// TIA Portal V20 export
TYPE "LBP_typeChanX"
TITLE = Channel interface / Interface de canal
// User data type for blocks LBP_Chan1 [DB21] .. LBP_Chan10 [DB30] / Type de données utilisateur pour les blocs LBP_Chan1 [DB21] .. LBP_Chan10 [DB30]
   STRUCT
      f0_0 : Bool;
      f0_1 : Bool;
      f0_2 : Bool;
      A_DRF : Bool;   // Activate DRF / Activer DRF
      A_SBL : Bool;   // Activate single block / Activer bloc par bloc
      A_M01 : Bool;   // Activate M01 / Activer M01
      A_DRY : Bool;   // Activate dry run feedrate / Activer avance marche d'essai
      f0_7 : Bool;
      A_Ref : Bool;   // Activate referencing / Activer référencement
      A_ProtZone : Bool;   // Enable protection zones / Activer zones de protection
      A_SynOff : Bool;   // Synchronous action off / Action synchrone désactivée
      A_TM_TimOut : Bool;   // Activate time-out (TM) / Activer timeout (TM)
      A_CLC_Stop : Bool;   // CLC stop / Stop CLC
      A_CLC_OR : Bool;   // CLC override / Correction CLC
      A_PLC_ActCompl : Bool;   // PLC action completed / Action AP terminée
      A_ProgTest : Bool;   // Activate program test / Activer test de programme
      A_SKP0 : Bool;   // Activate skip block \0 / Activer ignorer bloc \0
      A_SKP1 : Bool;   // Activate skip block \1 / Activer ignorer bloc \1
      A_SKP2 : Bool;   // Activate skip block \2 / Activer ignorer bloc \2
      A_SKP3 : Bool;   // Activate skip block \3 / Activer ignorer bloc \3
      A_SKP4 : Bool;   // Activate skip block \4 / Activer ignorer bloc \4
      A_SKP5 : Bool;   // Activate skip block \5 / Activer ignorer bloc \5
      A_SKP6 : Bool;   // Activate skip block \6 / Activer ignorer bloc \6
      A_SKP7 : Bool;   // Activate skip block \7 / Activer ignorer bloc \7
      A_StrokEnab : Bool;   // Stroke enable / Activer course
      A_ManStrokEnab : Bool;   // Manual stroke enable / Activation manuelle de la course
      A_StrokSup : Bool;   // Stroke suppression / Inhibition de course
      A_StrokDelayed : Bool;   // Stroke delayed / Course retardée
      A_StrokStop : Bool;   // Stroke not operating / Course inopérante
      A_ManRelStroke2 : Bool;   // Manual release of stroke 2 / Déblocage manuel de la course 2
      A3_6 : Bool;
      A3_7 : Bool;
      A_FD_OR : Byte;   // Feedrate override / Correction d'avance
      A_RT_OR : Byte;   // Rapid traverse override / Correction marche rapide
      A_FDdisable : Bool;   // Feed disable / Désactiver avance
      A_RIdisable : Bool;   // Read-in disable / Désactiver importation
      A_DeleteDTG : Bool;   // Delete distance to go / Effacer la distance restante à parcourir
      A_SP_Clear : Bool;   // Delete UP number of passes / Supprimer nombre UP de passes
      A_ProgAbort : Bool;   // Program level abort / Abandon niveau de programme
      A_F_Limit : Bool;   // Tool path feedrate limitation / Trajectoire d'outil limitation d'avance
      A_RT_ORA : Bool;   // Rapid traverse override active / Correction marche rapide active
      A_FD_ORA : Bool;   // Feedrate override active / Correction d'avance active
      A_NCStartDisabl : Bool;   // NC start disable / Désactiver Départ CN
      A_NCStart : Bool;   // NC start / Départ CN
      A_NCStopBlock : Bool;   // NC stop at block limit / Arrêt CN à la limite de bloc
      A_NCStop : Bool;   // NC stop / Arrêt CN
      A_NCStopASp : Bool;   // NC stop axes plus spindle / Arrêt CN axes et broche
      A_SuppStartLock : Bool;   // Suppress Start Lock / Inhiber blocage de démarrage
      A_CfgStopFunc : Bool;   // Activate configured stop function / Activer la fonction d'arrêt configuré
      A_Reset : Bool;   // Reset
      A_MRP : Array[1..10] of Bool;   // Activate machine-related protection zone [1..10] / Activer zone de protection référencée dans le SCM [1..10]
      A_CSP : Array[1..10] of Bool;   // Activate channel-specific protection zone [1..10] / Activer zone de protection spécifique au canal [1..10]
      A_Geo : Array[1..3] of Struct   // Control signals for geometry axis [1..3] / Signaux de commande pour axe géométrique [1..3]
         HW1 : Bool;   // Activate handwheel 1 / Activer manivelle 1
         HW2 : Bool;   // Activate handwheel 2 / Activer manivelle 2
         HW3 : Bool;   // Activate handwheel 3 / Activer manivelle 3
         FDStop : Bool;   // Feedrate stop / Arrêt avance
         Disabl : Bool;   // Traversing key disable / Désactiver la touche de déplacement
         RapidTrOR : Bool;   // Rapid traverse override / Correction marche rapide
         Minus : Bool;   // Traversing key minus / Touche de déplacement moins
         Plus : Bool;   // Traversing key plus / Touche de déplacement plus
         INC1 : Bool;   // INC 1
         INC10 : Bool;   // INC 10
         INC100 : Bool;   // INC 100
         INC1000 : Bool;   // INC 1000
         INC10000 : Bool;   // INC 10000
         INCVar : Bool;   // INC variable / Variable INC
         ContManTravel : Bool;   // Continuous manual travel / Mode manuel continu
         f1_7 : Bool;
         OEM : Byte;   // OEM signals / Signaux OEM
         InvHWDirOfRot : Bool;   // Invert handwheel direction of rotation / Inverser sens de rotation manivelle
         f3_1 : Bool;
         f3_2 : Bool;
         f3_3 : Bool;
         f3_4 : Bool;
         f3_5 : Bool;
         f3_6 : Bool;
         f3_7 : Bool;
      END_STRUCT;
      f24_0 : Bool;
      E_MMC_CfgStopFunc : Bool;   // HMI: configured stop function (CST) is selected / IHM : La fonction d'arrêt configuré (CST) est sélectionnée
      E_MMC_AtStopSetOvrZero : Bool;   // HMI: Set to 0% for stop override / IHM : à l'arrêt, régler la correction sur 0 %
      E_MMC_DRF : Bool;   // HMI DRF selected / HMI DRF sélectionné
      E_MMC_M01AssocNC : Bool;   // Select M01 associated with NC / Sélectionner M01 associé à CN
      E_MMC_M01 : Bool;   // HMI M01 selected / HMI M01 sélectionné
      E_MMC_DRY : Bool;   // HMI Dry-run feedrate selected / HMI Marche d'essai avance sélectionnée
      f24_7 : Bool;
      E_MMC_REPOSPM_0 : Bool;   // HMI REPOSPATHMODE 0
      E_MMC_REPOSPM_1 : Bool;   // HMI REPOSPATHMODE 1
      E_MMC_REPOSPM_2 : Bool;   // HMI REPOSPATHMODE 2
      E_MMC_FD_OR4RT_OR : Bool;   // HMI Feedrate override for rapid traverse selected / HMI Correction d'avance marche rapide sélectionnée
      E_MMC_REPOSMode : Bool;   // HMI REPOS MODE EDGE
      f25_5 : Bool;
      f25_6 : Bool;
      E_MMC_ProgTest : Bool;   // Program test selected / Test de programme sélectionné
      E_MMC_SKP0 : Bool;   // HMI skip block selected \0 / HMI Ignorer bloc sélectionné \0
      E_MMC_SKP1 : Bool;   // HMI skip block selected \1 / HMI Ignorer bloc sélectionné \1
      E_MMC_SKP2 : Bool;   // HMI skip block selected \2 / HMI Ignorer bloc sélectionné \2
      E_MMC_SKP3 : Bool;   // HMI skip block selected \3 / HMI Ignorer bloc sélectionné \3
      E_MMC_SKP4 : Bool;   // HMI skip block selected \4 / HMI Ignorer bloc sélectionné \4
      E_MMC_SKP5 : Bool;   // HMI skip block selected \5 / HMI Ignorer bloc sélectionné \5
      E_MMC_SKP6 : Bool;   // HMI skip block selected \6 / HMI Ignorer bloc sélectionné \6
      E_MMC_SKP7 : Bool;   // HMI skip block selected \7 / HMI Ignorer bloc sélectionné \7
      E_MMC_SKP8 : Bool;   // HMI skip block selected \8 / HMI Ignorer bloc sélectionné \8
      E_MMC_SKP9 : Bool;   // HMI skip block selected \9 / HMI Ignorer bloc sélectionné \9
      f27_2 : Bool;
      f27_3 : Bool;
      f27_4 : Bool;
      f27_5 : Bool;
      f27_6 : Bool;
      f27_7 : Bool;
      A_OEM : Byte;
      A_FixedFD1 : Bool;   // Activate fixed feedrate 1 / Activer l'avance fixe 1
      A_FixedFD2 : Bool;   // Activate fixed feedrate 2 / Activer l'avance fixe 2
      A_FixedFD3 : Bool;   // Activate fixed feedrate 3 / Activer l'avance fixe 3
      A_FixedFD4 : Bool;   // Activate fixed feedrate 4 / Activer l'avance fixe 4
      A_PTP_Travel : Bool;   // Activate PTP traversal / Activer déplacement PTP
      A_DisablWP_Counter : Bool;   // Deactivate workpiece counter / Désactiver compteur de pièces
      A_DisablWearMon : Bool;   // Deactivate wear monitoring / Désactiver surveillance d'usure
      A_DontDisablTool : Bool;   // Do not disable tool / Ne pas désactiver outil
      A_ContHW1 : Bool;   // Activate contour handwheel 1 / Activer manivelle de contour 1
      A_ContHW2 : Bool;   // Activate contour handwheel 2 / Activer manivelle de contour 2
      A_ContHW3 : Bool;   // Activate contour handwheel 3 / Activer manivelle de contour 3
      A_ContHWsim : Bool;   // Simulated contour handwheel on / Manivelle de contour simulée Marche
      A_ContHWneg : Bool;   // Contour handwheel neg. route / Manivelle de contour dépl. nég.
      A_NCKrelatedM01 : Bool;   // Activate NCK-related M01 / Activer M01 relatif à la NCK
      A_JOG_Circles : Bool;   // JOG in circles / JOG en cercles
      A_NoToolChangeCmd : Bool;   // No tool change commands / Aucun ordre de changement d'outil
      A_REPOSPM_0 : Bool;   // REPOSPATHMODE 0
      A_REPOSPM_1 : Bool;   // REPOSPATHMODE 1
      A_REPOSPM_2 : Bool;   // REPOSPATHMODE 2
      f31_3 : Bool;
      A_REPOSMode : Bool;   // REPOS MODE EDGE
      A_InvCHWDirOfRot : Bool;   // Inverting contour handwheel direction of rotation / Inversion du sens de rotation de la manivelle
      A_SKP8 : Bool;   // Activate skip block \8 / Activer ignorer bloc \8
      A_SKP9 : Bool;   // Activate skip block \9 / Activer ignorer bloc \9
      E_ExecExtern : Bool;   // Execution from external source active / Exécution à partir de source externe active
      f32_1 : Bool;
      f32_2 : Bool;
      E_ActBlock : Bool;   // Action block active / Bloc d'action actif
      E_BegBlock : Bool;   // Approach block active / Bloc d'accostage actif
      E_M01 : Bool;   // M0/M1 active / M0/M1 actif
      E_LastActBlock : Bool;   // Last action block active / Dernier bloc d'action actif
      f32_7 : Bool;
      E_Ref : Bool;   // Referencing active / Référencement actif
      E_OrieToolholder : Bool;   // Orientable toolholder active / Porte-outil orientable actif
      E_RevFD : Bool;   // Revolutional feedrate active / Avance par tour active
      E_HWOverlay : Bool;   // Handwheel override active / Correction manivelle active
      E_BlockSearch : Bool;   // Block search active / Recherche de blocs active
      E_M30 : Bool;   // M2/M30 active / M2/M30 actif
      E_Transform : Bool;   // Transformation active
      E_ProgTest : Bool;   // Program test active / Test de programme actif
      E_OEMChan : Byte;   // OEM channel signals feedback / Signalisation en retour signaux de canal OEM
      E_ProgRunning : Bool;   // Program running / Programme en cours d'exécution
      E_ProgWait : Bool;   // Program waiting / Programme en attente
      E_ProgStop : Bool;   // Program stopped / Programme arrêté
      E_ProgInterrupt : Bool;   // Program interrupted / Programme interrompu
      E_ProgAborted : Bool;   // Program aborted / Programme abandonné
      E_ChanActive : Bool;   // Channel active / Canal actif
      E_ChanInterrupt : Bool;   // Channel interrupted / Canal interrompu
      E_ChanReset : Bool;   // Channel reset / Reset canal
      E_StartReq : Bool;   // Start request / Demande de démarrage
      E_StopReq : Bool;   // Stop request / Demande d'arrêt
      E_AxesRef : Bool;   // All axes referenced / Référencer tous les axes
      E_AxesStop : Bool;   // All axes stationary / Tous les axes à l'arrêt
      E_IR_Activ : Bool;   // Interrupt processing active / Traitement d'interruption actif
      E_ChanRO : Bool;   // Channel ready for operation / Canal prêt à fonctionner
      E_NCKalarmChan : Bool;   // Channel-specific NCK alarm present / Alarme NCK spécifique à un canal présente
      E_NCKalarmStop : Bool;   // NCK alarm with processing stop present / Alarme NCK avec d'arrêt d'usinage présente
      E_CHW1 : Bool;   // Contour handwheel 1 on / Manivelle de contour 1
      E_CHW2 : Bool;   // Contour handwheel 2 on / Manivelle de contour 2
      E_CHW3 : Bool;   // Contour handwheel 3 on / Manivelle de contour 3
      E_CLC : Bool;   // CLC active / CLC actif
      E_CLCStopLL : Bool;   // CLC stopped lower limit / CLC arrêté limite inférieure
      E_CLCStopUL : Bool;   // CLC stopped upper limit / CLC arrêté limite supérieure
      E_RIEnabIgnored : Bool;   // Read-in enable is ignored / Activation Charger ignorée
      E_StopBlkEndSBLsuppr : Bool;   // Stop at block end with SBL is suppressed / Inhiber arrêt sur fin de bloc avec SBL
      E_StrokeEA : Bool;   // Stroke release active / Déblocage course actif
      E_AcknManStrokEnab : Bool;   // Acknowledgment of manual stroke release / Acquittement déblocage manuel de course
      f38_2 : Bool;
      f38_3 : Bool;
      f38_4 : Bool;
      f38_5 : Bool;
      f38_6 : Bool;
      f38_7 : Bool;
      E_ProtZoneNOK : Bool;   // Protection zones not guaranteed / Zones de protection non garanties
      E_NCalarmWithProgStop : Bool;   // NC alarm with program stop / Alarme CN avec arrêt du programme
      f39_2 : Bool;
      E_ReducedDynamicsActive : Bool;   // Reduced dynamics mode is active / Le mode de dynamique réduite est actif
      E_SblStopAtBlockEnd : Bool;   // Stop at block end due to single block / Arrêt en fin de bloc en raison du mode bloc par bloc
      E_InvCHWDirOfRot : Bool;   // Contour handwheel direction of rotation invert actively / Inversion active du sens de rotation manivelle de contour
      E_CfgStopFuncActive : Bool;   // Configured stop function is activated / La fonction d'arrêt configuré est activée
      E_CfgStopAtBlockEnd : Bool;   // Stop at block end due to configured stop / Arrêt en fin de bloc en raison de l'arrêt configuré
      E_Geo : Array[1..3] of Struct   // Status signals of geometry axis [1..3] / Signaux d'état de l'axe géométrique [1..3]
         HW1 : Bool;   // Handwheel 1 active / Manivelle 1 active
         HW2 : Bool;   // Handwheel 2 active / Manivelle 2 active
         HW3 : Bool;   // Handwheel 3 active / Manivelle 3 active
         f0_3 : Bool;
         TReqMinus : Bool;   // Travel requests minus / Demandes de déplacement moins
         TReqPlus : Bool;   // Travel requests plus / Demandes de déplacement plus
         TCMinus : Bool;   // Traverse command minus / Instruction de déplacement moins
         TCPlus : Bool;   // Traverse command plus / Instruction de déplacement plus
         INC1 : Bool;   // INC 1 active
         INC10 : Bool;   // INC 10 active
         INC100 : Bool;   // INC 100 active
         INC1000 : Bool;   // INC 1000 active
         INC10000 : Bool;   // INC 10000 active
         INCVar : Bool;   // INC variable active / Variable INC active
         ContManTravelAct : Bool;   // Continuous manual travel active / Mode manuel continu actif
         f1_7 : Bool;
         OEM : Byte;   // OEM signals / Signaux OEM
         InvHWDirOfRot : Bool;   // Handwheel direction of rotation invert actively / Inverser activement sens manivelle
         f3_1 : Bool;
         f3_2 : Bool;
         f3_3 : Bool;
         f3_4 : Bool;
         f3_5 : Bool;
         f3_6 : Bool;
         f3_7 : Bool;
         f4 : Byte;
      END_STRUCT;
      M1Change : Bool;   // M function 1 change / Fonction M 1 modification
      M2Change : Bool;   // M function 2 change / Fonction M 2 modification
      M3Change : Bool;   // M function 3 change / Fonction M 3 modification
      M4Change : Bool;   // M function 4 change / Fonction M 4 modification
      M5Change : Bool;   // M function 5 change / Fonction M 5 modification
      f58_5 : Bool;
      f58_6 : Bool;
      f58_7 : Bool;
      M1NDec : Bool;   // M function 1 not decoded / Fonction M 1 non décodée
      M2NDec : Bool;   // M function 2 not decoded / Fonction M 2 non décodée
      M3NDec : Bool;   // M function 3 not decoded / Fonction M 3 non décodée
      M4NDec : Bool;   // M function 4 not decoded / Fonction M 4 non décodée
      M5NDec : Bool;   // M function 5 not decoded / Fonction M 5 non décodée
      f59_5 : Bool;
      f59_6 : Bool;
      f59_7 : Bool;
      S1Change : Bool;   // S function 1 change / Fonction S 1 modification
      S2Change : Bool;   // S function 2 change / Fonction S 2 modification
      S3Change : Bool;   // S function 3 change / Fonction S 3 modification
      f60_3 : Bool;
      S1Quick : Bool;   // S function 1 quick / Fonction S 1 rapide
      S2Quick : Bool;   // S function 2 quick / Fonction S 2 rapide
      S3Quick : Bool;   // S function 3 quick / Fonction S 3 rapide
      f60_7 : Bool;
      T1Change : Bool;   // T function 1 change / Fonction T 1 modification
      T2Change : Bool;   // T function 2 change / Fonction T 2 modification
      T3Change : Bool;   // T function 3 change / Fonction T 3 modification
      f61_3 : Bool;
      T1Quick : Bool;   // T function 1 quick / Fonction T 1 rapide
      T2Quick : Bool;   // T function 2 quick / Fonction T 2 rapide
      T3Quick : Bool;   // T function 3 quick / Fonction T 3 rapide
      f61_7 : Bool;
      D1Change : Bool;   // D function 1 change / Fonction D 1 modification
      D2Change : Bool;   // D function 2 change / Fonction D 2 modification
      D3Change : Bool;   // D function 3 change / Fonction D 3 modification
      f62_3 : Bool;
      D1Quick : Bool;   // D function 1 quick / Fonction D 1 rapide
      D2Quick : Bool;   // D function 2 quick / Fonction D 2 rapide
      D3Quick : Bool;   // D function 3 quick / Fonction D 3 rapide
      f62_7 : Bool;
      EChange : Bool;   // E function change / Fonction E modification
      f63_1 : Bool;
      f63_2 : Bool;
      f63_3 : Bool;
      EQuick : Bool;   // E function quick / Fonction E rapide
      f63_5 : Bool;
      f63_6 : Bool;
      f63_7 : Bool;
      H1Change : Bool;   // H function 1 change / Fonction H 1 modification
      H2Change : Bool;   // H function 2 change / Fonction H 2 modification
      H3Change : Bool;   // H function 3 change / Fonction H 3 modification
      f64_3 : Bool;
      H1Quick : Bool;   // H function 1 quick / Fonction H 1 rapide
      H2Quick : Bool;   // H function 2 quick / Fonction H 2 rapide
      H3Quick : Bool;   // H function 3 quick / Fonction H 3 rapide
      f64_7 : Bool;
      F1Change : Bool;   // F function 1 change / Fonction F 1 modification
      F2Change : Bool;   // F function 2 change / Fonction F 2 modification
      F3Change : Bool;   // F function 3 change / Fonction F 3 modification
      F4Change : Bool;   // F function 4 change / Fonction F 4 modification
      F5Change : Bool;   // F function 5 change / Fonction F 5 modification
      F6Change : Bool;   // F function 6 change / Fonction F 6 modification
      f65_6 : Bool;
      f65_7 : Bool;
      M1Quick : Bool;   // M function 1 quick / Fonction M 1 rapide
      M2Quick : Bool;   // M function 2 quick / Fonction M 2 rapide
      M3Quick : Bool;   // M function 3 quick / Fonction M 3 rapide
      M4Quick : Bool;   // M function 4 quick / Fonction M 4 rapide
      M5Quick : Bool;   // M function 5 quick / Fonction M 5 rapide
      f66_5 : Bool;
      f66_6 : Bool;
      f66_7 : Bool;
      F1Quick : Bool;   // F function 1 quick / Fonction F 1 rapide
      F2Quick : Bool;   // F function 2 quick / Fonction F 2 rapide
      F3Quick : Bool;   // F function 3 quick / Fonction F 3 rapide
      F4Quick : Bool;   // F function 4 quick / Fonction F 4 rapide
      F5Quick : Bool;   // F function 5 quick / Fonction F 5 rapide
      F6Quick : Bool;   // F function 6 quick / Fonction F 6 rapide
      f67_6 : Bool;
      f67_7 : Bool;
      ExtM1 : Int;   // Extended address M function 1 (16 bit INT) / Fonction M à adresse étendue 1 (16 bits INT)
      M1 : DInt;   // M function 1 (DInt) / Fonction M 1 (DInt)
      ExtM2 : Int;   // Extended address M function 1 (16 bit INT) / Fonction M à adresse étendue 1 (16 bits INT)
      M2 : DInt;   // M function 2 (DInt) / Fonction M 2 (DInt)
      ExtM3 : Int;   // Extended address M function 1 (16 bit INT) / Fonction M à adresse étendue 1 (16 bits INT)
      M3 : DInt;   // M function 3 (DInt) / Fonction M 3 (DInt)
      ExtM4 : Int;   // Extended address M function 1 (16 bit INT) / Fonction M à adresse étendue 1 (16 bits INT)
      M4 : DInt;   // M function 4 (DInt) / Fonction M 4 (DInt)
      ExtM5 : Int;   // Extended address M function 1 (16 bit INT) / Fonction M à adresse étendue 1 (16 bits INT)
      M5 : DInt;   // M function 5 (DInt) / Fonction M 5 (DInt)
      ExtS1 : Int;   // Extended address S function 1 (16 bit INT) / Fonction S à adresse étendue 1 (16 bits INT)
      S1 : Real;   // S function 1 (REAL) / Fonction S 1 (REAL)
      ExtS2 : Int;   // Extended address S function 2 (16 bit INT) / Fonction S à adresse étendue 2 (16 bits INT)
      S2 : Real;   // S function 2 (REAL) / Fonction S 2 (REAL)
      ExtS3 : Int;   // Extended address S function 3 (16 bit INT) / Fonction S à adresse étendue 3 (16 bits INT)
      S3 : Real;   // S function 3 (REAL) / Fonction S 3 (REAL)
      ExtT1 : Int;   // Extended address T function 1 (16 bit INT)T : DINT; //T function (DInt)f122 : INT;f124 : INT;f126 : INT; //Change in case of 8-digit T function / Fonction T à adresse étendue 1 (16 Bit INT)T : DINT; //fonction T (DInt)f122 : INT;f124 : INT;f126 : INT; //Modifier pour une fonction T à 8 chiffres
      T1 : Int;   // T function 1 (INT) / Fonction T 1 (INT)
      ExtT2 : Int;   // Extended address T function 2 (16 bit INT) / Fonction T à adresse étendue 2 (16 bits INT)
      T2 : Int;   // T function 2 (INT) / Fonction T 2 (INT)
      ExtT3 : Int;   // Extended address T function 3 (16 bit INT) / Fonction T à adresse étendue 3 (16 bits INT)
      T3 : Int;   // T function 3 (INT) / Fonction T 3 (INT)
      ExtD1 : Byte;   // Extended address D function 1 (8 bit INT)D : INT;f132 : INT; //Change in case of 5-digit D function / Fonction D à adresse étendue 1 (8 bits INT)D : INT;f132 : INT; //Modifier pour une fonction D à 5 chiffres
      D1 : Byte;   // D function 1 (8 bit INT) / Fonction D 1 (8 bits INT)
      ExtD2 : Byte;   // Extended address D function 2 (8 bit INT) / Fonction D à adresse étendue 2 (8 bits INT)
      D2 : Byte;   // D function 2 (8 bit INT) / Fonction D 2 (8 bits INT)
      ExtD3 : Byte;   // Extended address D function 3 (8 bit INT) / Fonction D à adresse étendue 3 (8 bits INT)
      D3 : Byte;   // D function 3 (8 bit INT) / Fonction D 3 (8 bits INT)
      ExtE : Int;   // Extended address D function 3 (16 bit INT) / Fonction D à adresse étendue 3 (16 bits INT)
      "E" : Real;   // E function (REAL) / Fonction E (REAL)
      ExtH1 : Int;   // Extended address H function 1 (16 bit INT) / Fonction H à adresse étendue 1 (16 bits INT)
      H1 : Real;   // H function 1 (REAL), DInt also in DBD396 / Fonction H 1 (REAL), DInt également dans DBD396
      ExtH2 : Int;   // Extended address H function 2 (16 bit INT) / Fonction H à adresse étendue 2 (16 bits INT)
      H2 : Real;   // H function 2 (REAL), DInt also in DBD400 / Fonction H 2 (REAL), DInt également dans DBD400
      ExtH3 : Int;   // Extended address H function 3 (16 bit INT) / Fonction H à adresse étendue 3 (16 bits INT)
      H3 : Real;   // H function 3 (REAL), DInt also in DBD404 / Fonction H 3 (REAL), DInt également dans DBD404
      ExtF1 : Int;   // Extended address F function 1 (16 bit INT) / Fonction F à adresse étendue 1 (16 bits INT)
      F1 : Real;   // F function 1 (REAL) / Fonction F 1 (REAL)
      ExtF2 : Int;   // Extended address F function 2 (16 bit INT) / Fonction F à adresse étendue 2 (16 bits INT)
      F2 : Real;   // F function 2 (REAL) / Fonction F 2 (REAL)
      ExtF3 : Int;   // Extended address F function 3 (16 bit INT) / Fonction F à adresse étendue 3 (16 bits INT)
      F3 : Real;   // F function 3 (REAL) / Fonction F 3 (REAL)
      ExtF4 : Int;   // Extended address F function 4 (16 bit INT) / Fonction F à adresse étendue 4 (16 bits INT)
      F4 : Real;   // F function 4 (REAL) / Fonction F 4 (REAL)
      ExtF5 : Int;   // Extended address F function 5 (16 bit INT) / Fonction F à adresse étendue 5 (16 bits INT)
      F5 : Real;   // F function 5 (REAL) / Fonction F 5 (REAL)
      ExtF6 : Int;   // Extended address F function 6 (16 bit INT) / Fonction F à adresse étendue 6 (16 bits INT)
      F6 : Real;   // F function 6 (REAL) / Fonction F 6 (REAL)
      MDyn : Array[0..99] of Bool;   // Dynamic M functions [0..99] / Fonctions M dynamiques [0..99]
      GAct : Array[1..64] of Byte;   // Active G function of group [1..64] / Fonction G active du groupe [1..64]
      E_MRPactivated : Array[1..10] of Bool;   // Machine-related protection zone [1..10] preactivated / Zone de protection référencée dans le SCM [1..10] préactivé
      E_CSPactivated : Array[1..10] of Bool;   // Channel-specific protection zone [1..10] preactivated / Zone de protection spécifique au canal [1..10] préactivée
      E_MRPViolated : Array[1..10] of Bool;   // Machine-related protection zone [1..10] violated / Zone de protection référencée dans le SCM [1..10] dépassée
      E_CSPViolated : Array[1..10] of Bool;   // Channel-specific protection zone [1..10] violated from P4 on / Zone de protection spécifique au canal [1..10] dépassée à partir de P4
      f_280_0 : Bool;
      A_Str_Synon : Bool;   // Request of syn.action to NCK / Demande d'action synchrone vers NCK
      f_280_2 : Bool;
      f_280_3 : Bool;
      f_280_4 : Bool;
      f_280_5 : Bool;
      f_280_6 : Bool;
      f_280_7 : Bool;
      f_281_0 : Bool;
      A_Str_Synfrom : Bool;   // Request syn.action from NCK / Demande d'action synchrone depuis NCK
      f_281_2 : Bool;
      f_281_3 : Bool;
      f_281_4 : Bool;
      f_281_5 : Bool;
      f_281_6 : Bool;
      f_281_7 : Bool;
      f_282 : Int;
      f_284 : Int;
      f_286 : Int;
      f_288 : Int;
      f_290 : Int;
      f_292 : Int;
      f_294 : Int;
      f_296 : Int;
      f_298 : Int;
      A_SynDisabl : Array[1..64] of Bool;   // Disable synchronous actions / Désactiver actions synchrones
      E_SynDisabled : Array[1..64] of Bool;   // Synchronous actions disabled / Actions synchrones désactivées
      E_G00 : Bool;   // Active G functions / Fonctions G actives
      f316_1 : Bool;
      f316_2 : Bool;
      f316_3 : Bool;
      f316_4 : Bool;
      f316_5 : Bool;
      f316_6 : Bool;
      f316_7 : Bool;
      E_ExtLang : Bool;   // External language mode active / Mode de langage externe actif
      E_WS_Setp : Bool;   // Workpiece setpoint reached / Consigne pièce atteinte
      f317_2 : Bool;
      f317_3 : Bool;
      f317_4 : Bool;
      E_DriveTest : Bool;   // Travel request drive test / Demande de déplacement test d'entraînement
      E_PTP_Travel : Bool;   // PTP travel active / Déplacement PTP actif
      E_ToolMissing : Bool;   // Tool missing / Outil manquant
      E_ASUP_Stop : Bool;   // ASUP stopped / ASUP arrêté
      E_SearchAct : Bool;   // Search active / Recherche active
      E_TOFF : Bool;   // TOFF active / TOFF actif
      E_TOFFmovem : Bool;   // TOFF motion active / Déplacement TOFF actif
      E_StopDelayed : Bool;   // Stop delayed / Arrêt temporisé
      E_AssM01 : Bool;   // Associated M01 active / M01 associé actif
      E_DRY : Bool;   // Dry-run feedrate active / Marche d'essai avance active
      E_Overstore : Bool;   // Overstore active / Overstore actif
      E_REPOS_EdgeAckn : Bool;   // REPOS MODE EDGE ACKN
      E_REPOS_PMode0 : Bool;   // REPOS Path Mode Ackn 0
      E_REPOS_PMode1 : Bool;   // REPOS Path Mode Ackn 1
      E_REPOS_PMode2 : Bool;   // REPOS Path Mode Ackn 2
      E_DelayFTS : Bool;   // Delay FTS / Temporisation FTS
      E_REPOS_DEFERRA : Bool;   // REPOS DEFERRA L Chan
      E_Stop_NoDelayR : Bool;   // Stop-delay area not accepted / Plage de temporisation d'arrêt non acceptée
      E_NoToolChangeCmd : Bool;   // No tool change command active / Aucun ordre de changement d'outil actif
      A_Ori : Array[1..3] of Struct   // Control signals for orientation axes [1..3] / Signaux de commande pour axes d'orientation [1..3]
         HW1 : Bool;   // Activate handwheel 1 / Activer manivelle 1
         HW2 : Bool;   // Activate handwheel 2 / Activer manivelle 2
         HW3 : Bool;   // Activate handwheel 3 / Activer manivelle 3
         FDStop : Bool;   // Feedrate stop / Arrêt avance
         Disabl : Bool;   // Traversing key lock / Verrouiller touche de déplacement
         RapidTrOR : Bool;   // Rapid traverse override / Correction marche rapide
         Minus : Bool;   // Traversing key minus / Touche de déplacement moins
         Plus : Bool;   // Traversing key plus / Touche de déplacement plus
         INC1 : Bool;   // INC 1 active
         INC10 : Bool;   // INC 10 active
         INC100 : Bool;   // INC 100 active
         INC1000 : Bool;   // INC 1000 active
         INC10000 : Bool;   // INC 10000 active
         INCVar : Bool;   // INC variable active / Variable INC active
         OEM : Byte;   // OEM signals / Signaux OEM
         InvHWDirOfRot : Bool;   // Inverting handwheel direction of rotation / Inverser sens de rotation manivelle
         f3_1 : Bool;
         f3_2 : Bool;
         f3_3 : Bool;
         f3_4 : Bool;
         f3_5 : Bool;
         f3_6 : Bool;
         f3_7 : Bool;
      END_STRUCT;
      E_Ori : Array[1..3] of Struct   // Control signals for orientation axes [1..3] / Signaux de commande pour axes d'orientation [1..3]
         HW1 : Bool;   // Handwheel 1 active / Manivelle 1 active
         HW2 : Bool;   // Handwheel 2 active / Manivelle 2 active
         HW3 : Bool;   // Handwheel 3 active / Manivelle 3 active
         f0_3 : Bool;
         TReqMinus : Bool;   // Travel requests minus / Demandes de déplacement moins
         TReqPlus : Bool;   // Travel requests plus / Demandes de déplacement plus
         TCMinus : Bool;   // Traverse command minus / Instruction de déplacement moins
         TCPlus : Bool;   // Traverse command plus / Instruction de déplacement plus
         INC1 : Bool;   // INC 1 active
         INC10 : Bool;   // INC 10 active
         INC100 : Bool;   // INC 100 active
         INC1000 : Bool;   // INC 1000 active
         INC10000 : Bool;   // INC 10000 active
         INCVar : Bool;   // INC variable active / Variable INC active
         OEM : Byte;   // OEM signals / Signaux OEM
         InvHWDirOfRot : Bool;   // Handwheel direction of rotation invert actively / Inverser activement sens manivelle
         f3_1 : Bool;
         f3_2 : Bool;
         f3_3 : Bool;
         f3_4 : Bool;
         f3_5 : Bool;
         f3_6 : Bool;
         f3_7 : Bool;
      END_STRUCT;
      E_TPrewarnLimit : Bool;   // Tool prewarn limit reached / Seuil de préavis outil atteint
      E_TLimit : Bool;   // Tool limit reached / Limite d'outil atteinte
      E_TNewRepl : Bool;   // Transition to new replacement tool / Transition vers nouvel outil de remplacement
      E_TLastRepl : Bool;   // Last replacement tool of the tool group / Dernier outil de remplacement du groupe d'outils
      f344_4 : Bool;
      f344_5 : Bool;
      f344_6 : Bool;
      f344_7 : Bool;
      f345 : Byte;
      f346 : Byte;
      f347 : Byte;
      E_TNoPrewarnLimit : DInt;   // T number for tool prewarn limit / Numéro d'outil pour seuil de préavis outil
      E_TNoLimit : DInt;   // T number for tool limit / Numéro d'outil pour limite d'outil
      E_TNoNewRepl : DInt;   // T number of the new replacement tool / Numéro d'outil du nouvel outil de remplacement
      E_TNoLastRepl : DInt;   // T number of the last replacement tool / Numéro d'outil du dernier outil de remplacement
      E_Cycle_Sig : Array[0..15] of Bool;   // Cycles input signals / Signaux d'entrée des cycles
      A_Cycle_Sig : Array[0..15] of Bool;   // Cycles output signals / Signaux de sortie des cycles
      E_OEM_TechnoSig : Array[0..31] of Bool;   // OEM Techno input signals / Signaux d'entrée techno OEM
      A_OEM_TechnoSig : Array[0..31] of Bool;   // OEM Techno output signals / Signaux de sortie techno OEM
      E_ProgEvent_Start : Bool;   // Active Prog-Event: Start / Prog-Event actif : Démarrage
      E_ProgEvent_M30 : Bool;   // Active Prog-Event: M30 / Prog-Event actif : M30
      E_ProgEvent_Reset : Bool;   // Active Prog-Event: Start / Prog-Event actif : Démarrage
      E_ProgEvent_PowerOn : Bool;   // Active Prog-Event: Power on / Prog-Event actif : Mise sous tension
      E_ProgEvent_SearchRun : Bool;   // Active Prog-Event: Search / Prog-Event actif : Recherche
      f376_5 : Bool;
      f376_6 : Bool;
      f376_7 : Bool;
      E_CollCheckStop : Bool;   // Stop of Collision Check / Arrêt du contrôle de collision
      E_StopCondition : Bool;   // Stop Condition / Condition d'arrêt
      f377_2 : Bool;
      f377_3 : Bool;
      E_JogRetract : Bool;   // JOG Retract active / Retrait JOG actif
      E_RetractData : Bool;   // Retract data available / Données de retrait disponibles
      E_JOG_Circles : Bool;   // JOG in circles / JOG en cercles
      f377_7 : Bool;
      E_AnyAsup : Bool;   // AnyASUP activ / AnyASUP actif
      E_SilentAsup : Bool;   // Silent ASUP active / ASUP silencieux actif
      f378_2 : Bool;
      f378_3 : Bool;
      f378_4 : Bool;
      f378_5 : Bool;
      f378_6 : Bool;
      f378_7 : Bool;
      f379 : Byte;
      f380 : Array[0..31] of Bool;   // Reserved / Réservé
      A_ProgJump : Bool;   // Control program jump / Saut programme de commande
      f384_1 : Bool;
      f384_2 : Bool;
      f384_3 : Bool;
      f384_4 : Bool;
      f384_5 : Bool;
      f384_6 : Bool;
      f384_7 : Bool;
      A_InKeyG1 : Bool;   // Grinding signal 1 / Signal rectification 1
      A_InKeyG2 : Bool;   // Grinding signal 2 / Signal rectification 2
      A_InKeyG3 : Bool;   // Grinding signal 3 / Signal rectification 3
      A_InKeyG4 : Bool;   // Grinding signal 4 / Signal rectification 4
      A_InKeyG5 : Bool;   // Grinding signal 5 / Signal rectification 5
      A_InKeyG6 : Bool;   // Grinding signal 6 / Signal rectification 6
      A_InKeyG7 : Bool;   // Grinding signal 7 / Signal rectification 7
      A_InKeyG8 : Bool;   // Grinding signal 8 / Signal rectification 8
      A_InKeyGEn1 : Bool;   // Enable grinding signal 1 / Activer signal rectification 1
      A_InKeyGEn2 : Bool;   // Enable grinding signal 2 / Activer signal rectification 2
      A_InKeyGEn3 : Bool;   // Enable grinding signal 3 / Activer signal rectification 3
      A_InKeyGEn4 : Bool;   // Enable grinding signal 4 / Activer signal rectification 4
      A_InKeyGEn5 : Bool;   // Enable grinding signal 5 / Activer signal rectification 5
      A_InKeyGEn6 : Bool;   // Enable grinding signal 6 / Activer signal rectification 6
      A_InKeyGEn7 : Bool;   // Enable grinding signal 7 / Activer signal rectification 7
      A_InKeyGEn8 : Bool;   // Enable grinding signal 8 / Activer signal rectification 8
      A_InKeyGRunIn1 : Bool;   // Run grinding function 1 / Exécuter fonction de rectification 1
      A_InKeyGRunIn2 : Bool;   // Run grinding function 2 / Exécuter fonction de rectification 2
      A_InKeyGRunIn3 : Bool;   // Run grinding function 3 / Exécuter fonction de rectification 3
      A_InKeyGRunIn4 : Bool;   // Run grinding function 4 / Exécuter fonction de rectification 4
      A_InKeyGRunIn5 : Bool;   // Run grinding function 5 / Exécuter fonction de rectification 5
      A_InKeyGRunIn6 : Bool;   // Run grinding function 6 / Exécuter fonction de rectification 6
      A_InKeyGRunIn7 : Bool;   // Run grinding function 7 / Exécuter fonction de rectification 7
      A_InKeyGRunIn8 : Bool;   // Run grinding function 8 / Exécuter fonction de rectification 8
      E_TransformNo : Byte;   // Active transformation number / Numéro de la transformation active
      f389 : Byte;
      E_InKeyGIsEn1 : Bool;   // Grinding signal 1 enabled / Signal rectification 1 activé
      E_InKeyGIsEn2 : Bool;   // Grinding signal 2 enabled / Signal rectification 2 activé
      E_InKeyGIsEn3 : Bool;   // Grinding signal 3 enabled / Signal rectification 3 activé
      E_InKeyGIsEn4 : Bool;   // Grinding signal 4 enabled / Signal rectification 4 activé
      E_InKeyGIsEn5 : Bool;   // Grinding signal 5 enabled / Signal rectification 5 activé
      E_InKeyGIsEn6 : Bool;   // Grinding signal 6 enabled / Signal rectification 6 activé
      E_InKeyGIsEn7 : Bool;   // Grinding signal 7 enabled / Signal rectification 7 activé
      E_InKeyGIsEn8 : Bool;   // Grinding signal 8 enabled / Signal rectification 8 activé
      E_InKeyGRunOut1 : Bool;   // NCK status of grinding function 1 / État NCK fonction de rectification 1
      E_InKeyGRunOut2 : Bool;   // NCK status of grinding function 3 / État NCK fonction de rectification 3
      E_InKeyGRunOut3 : Bool;   // NCK status of grinding function 3 / État NCK fonction de rectification 3
      E_InKeyGRunOut4 : Bool;   // NCK status of grinding function 4 / État NCK fonction de rectification 4
      E_InKeyGRunOut5 : Bool;   // NCK status of grinding function 5 / État NCK fonction de rectification 5
      E_InKeyGRunOut6 : Bool;   // NCK status of grinding function 6 / État NCK fonction de rectification 6
      E_InKeyGRunOut7 : Bool;   // NCK status of grinding function 7 / État NCK fonction de rectification 7
      E_InKeyGRunOut8 : Bool;   // NCK status of grinding function 8 / État NCK fonction de rectification 8
      E_CART_JOG_MODE : Byte;   // Coordinate system for Cartesian jog traverse / Système de coordonnées pour déplacement cartésien en mode JOG
      f393 : Byte;
      f394 : Byte;
      f395 : Byte;
      H1_DInt : DInt;   // H Function 1 (DInt) / Fonction H 1 (DInt)
      H2_DInt : DInt;   // H Function 2 (DInt) / Fonction H 2 (DInt)
      H3_DInt : DInt;   // H Function 3 (DInt) / Fonction H 3 (DInt)
      E_AxisSelType : Byte;   // 0: MachAxis, 1: GeoAxis
      E_AxisSelAxis : Byte;   // Axis number / Numéro d'axe
      E_AxisSelRequest : Bool;   // Axis selection (touch) / Sélection d'axe (touche)
      f410_1 : Bool;
      f410_2 : Bool;
      f410_3 : Bool;
      f410_4 : Bool;
      f410_5 : Bool;
      f410_6 : Bool;
      f410_7 : Bool;
      f411 : Byte;
      A_AxisSelTypeActive : Byte;   // 0: MachAxis, 1: GeoAxis (return) / 0: MachAxis, 1: GeoAxis (retour)
      A_AxisSelAxisActive : Byte;   // Axis number (return) / Numéro d'axe (retour)
   END_STRUCT;
   // // A_Geo[2].HW1 : Activate handwheel 1 / Activer manivelle 1
   // // A_Geo[3].HW1 : Activate handwheel 1 / Activer manivelle 1
   // // A_Geo[2].HW2 : Activate handwheel 2 / Activer manivelle 2
   // // A_Geo[3].HW2 : Activate handwheel 2 / Activer manivelle 2
   // // A_Geo[2].HW3 : Activate handwheel 3 / Activer manivelle 3
   // // A_Geo[3].HW3 : Activate handwheel 3 / Activer manivelle 3
   // // A_Geo[2].FDStop : Feedrate stop / Arrêt avance
   // // A_Geo[3].FDStop : Feedrate stop / Arrêt avance
   // // A_Geo[2].Disabl : Traversing key disable / Désactiver la touche de déplacement
   // // A_Geo[3].Disabl : Traversing key disable / Désactiver la touche de déplacement
   // // A_Geo[2].RapidTrOR : Rapid traverse override / Correction marche rapide
   // // A_Geo[3].RapidTrOR : Rapid traverse override / Correction marche rapide
   // // A_Geo[2].Minus : Traversing key minus / Touche de déplacement moins
   // // A_Geo[3].Minus : Traversing key minus / Touche de déplacement moins
   // // A_Geo[2].Plus : Traversing key plus / Touche de déplacement plus
   // // A_Geo[3].Plus : Traversing key plus / Touche de déplacement plus
   // // A_Geo[2].INC1 : INC 1
   // // A_Geo[3].INC1 : INC 1
   // // A_Geo[2].INC10 : INC 10
   // // A_Geo[3].INC10 : INC 10
   // // A_Geo[2].INC100 : INC 100
   // // A_Geo[3].INC100 : INC 100
   // // A_Geo[2].INC1000 : INC 1000
   // // A_Geo[3].INC1000 : INC 1000
   // // A_Geo[2].INC10000 : INC 10000
   // // A_Geo[3].INC10000 : INC 10000
   // // A_Geo[2].INCVar : INC variable / Variable INC
   // // A_Geo[3].INCVar : INC variable / Variable INC
   // // A_Geo[2].ContManTravel : Continuous manual travel / Mode manuel continu
   // // A_Geo[3].ContManTravel : Continuous manual travel / Mode manuel continu
   // // A_Geo[2].OEM : OEM signals / Signaux OEM
   // // A_Geo[3].OEM : OEM signals / Signaux OEM
   // // A_Geo[2].InvHWDirOfRot : Invert handwheel direction of rotation / Inverser sens de rotation manivelle
   // // A_Geo[3].InvHWDirOfRot : Invert handwheel direction of rotation / Inverser sens de rotation manivelle
   // // A_Geo[1] : Control signals for geometry axis [1..3] / Signaux de commande pour axe géométrique [1..3]
   // // A_Geo[2] : Control signals for geometry axis [1..3] / Signaux de commande pour axe géométrique [1..3]
   // // A_Geo[3] : Control signals for geometry axis [1..3] / Signaux de commande pour axe géométrique [1..3]
   // // E_Geo[2].HW1 : Handwheel 1 active / Manivelle 1 active
   // // E_Geo[3].HW1 : Handwheel 1 active / Manivelle 1 active
   // // E_Geo[2].HW2 : Handwheel 2 active / Manivelle 2 active
   // // E_Geo[3].HW2 : Handwheel 2 active / Manivelle 2 active
   // // E_Geo[2].HW3 : Handwheel 3 active / Manivelle 3 active
   // // E_Geo[3].HW3 : Handwheel 3 active / Manivelle 3 active
   // // E_Geo[2].TReqMinus : Travel requests minus / Demandes de déplacement moins
   // // E_Geo[3].TReqMinus : Travel requests minus / Demandes de déplacement moins
   // // E_Geo[2].TReqPlus : Travel requests plus / Demandes de déplacement plus
   // // E_Geo[3].TReqPlus : Travel requests plus / Demandes de déplacement plus
   // // E_Geo[2].TCMinus : Traverse command minus / Instruction de déplacement moins
   // // E_Geo[3].TCMinus : Traverse command minus / Instruction de déplacement moins
   // // E_Geo[2].TCPlus : Traverse command plus / Instruction de déplacement plus
   // // E_Geo[3].TCPlus : Traverse command plus / Instruction de déplacement plus
   // // E_Geo[2].INC1 : INC 1 active
   // // E_Geo[3].INC1 : INC 1 active
   // // E_Geo[2].INC10 : INC 10 active
   // // E_Geo[3].INC10 : INC 10 active
   // // E_Geo[2].INC100 : INC 100 active
   // // E_Geo[3].INC100 : INC 100 active
   // // E_Geo[2].INC1000 : INC 1000 active
   // // E_Geo[3].INC1000 : INC 1000 active
   // // E_Geo[2].INC10000 : INC 10000 active
   // // E_Geo[3].INC10000 : INC 10000 active
   // // E_Geo[2].INCVar : INC variable active / Variable INC active
   // // E_Geo[3].INCVar : INC variable active / Variable INC active
   // E_Geo[1].ContManTravelAct := false;
   // // E_Geo[2].ContManTravelAct : Continuous manual travel active / Mode manuel continu actif
   // // E_Geo[3].ContManTravelAct : Continuous manual travel active / Mode manuel continu actif
   // E_Geo[1].f1_7 := false;
   // // E_Geo[2].OEM : OEM signals / Signaux OEM
   // // E_Geo[3].OEM : OEM signals / Signaux OEM
   // // E_Geo[2].InvHWDirOfRot : Handwheel direction of rotation invert actively / Inverser activement sens manivelle
   // // E_Geo[3].InvHWDirOfRot : Handwheel direction of rotation invert actively / Inverser activement sens manivelle
   // // E_Geo[1] : Status signals of geometry axis [1..3] / Signaux d'état de l'axe géométrique [1..3]
   // // E_Geo[2] : Status signals of geometry axis [1..3] / Signaux d'état de l'axe géométrique [1..3]
   // // E_Geo[3] : Status signals of geometry axis [1..3] / Signaux d'état de l'axe géométrique [1..3]
   // // A_Ori[2].HW1 : Activate handwheel 1 / Activer manivelle 1
   // // A_Ori[3].HW1 : Activate handwheel 1 / Activer manivelle 1
   // // A_Ori[2].HW2 : Activate handwheel 2 / Activer manivelle 2
   // // A_Ori[3].HW2 : Activate handwheel 2 / Activer manivelle 2
   // // A_Ori[2].HW3 : Activate handwheel 3 / Activer manivelle 3
   // // A_Ori[3].HW3 : Activate handwheel 3 / Activer manivelle 3
   // // A_Ori[2].FDStop : Feedrate stop / Arrêt avance
   // // A_Ori[3].FDStop : Feedrate stop / Arrêt avance
   // // A_Ori[2].Disabl : Traversing key lock / Verrouiller touche de déplacement
   // // A_Ori[3].Disabl : Traversing key lock / Verrouiller touche de déplacement
   // // A_Ori[2].RapidTrOR : Rapid traverse override / Correction marche rapide
   // // A_Ori[3].RapidTrOR : Rapid traverse override / Correction marche rapide
   // // A_Ori[2].Minus : Traversing key minus / Touche de déplacement moins
   // // A_Ori[3].Minus : Traversing key minus / Touche de déplacement moins
   // // A_Ori[2].Plus : Traversing key plus / Touche de déplacement plus
   // // A_Ori[3].Plus : Traversing key plus / Touche de déplacement plus
   // // A_Ori[2].INC1 : INC 1 active
   // // A_Ori[3].INC1 : INC 1 active
   // // A_Ori[2].INC10 : INC 10 active
   // // A_Ori[3].INC10 : INC 10 active
   // // A_Ori[2].INC100 : INC 100 active
   // // A_Ori[3].INC100 : INC 100 active
   // // A_Ori[2].INC1000 : INC 1000 active
   // // A_Ori[3].INC1000 : INC 1000 active
   // // A_Ori[2].INC10000 : INC 10000 active
   // // A_Ori[3].INC10000 : INC 10000 active
   // // A_Ori[2].INCVar : INC variable active / Variable INC active
   // // A_Ori[3].INCVar : INC variable active / Variable INC active
   // // A_Ori[2].OEM : OEM signals / Signaux OEM
   // // A_Ori[3].OEM : OEM signals / Signaux OEM
   // // A_Ori[2].InvHWDirOfRot : Inverting handwheel direction of rotation / Inverser sens de rotation manivelle
   // // A_Ori[3].InvHWDirOfRot : Inverting handwheel direction of rotation / Inverser sens de rotation manivelle
   // // A_Ori[1] : Control signals for orientation axes [1..3] / Signaux de commande pour axes d'orientation [1..3]
   // // A_Ori[2] : Control signals for orientation axes [1..3] / Signaux de commande pour axes d'orientation [1..3]
   // // A_Ori[3] : Control signals for orientation axes [1..3] / Signaux de commande pour axes d'orientation [1..3]
   // // E_Ori[2].HW1 : Handwheel 1 active / Manivelle 1 active
   // // E_Ori[3].HW1 : Handwheel 1 active / Manivelle 1 active
   // // E_Ori[2].HW2 : Handwheel 2 active / Manivelle 2 active
   // // E_Ori[3].HW2 : Handwheel 2 active / Manivelle 2 active
   // // E_Ori[2].HW3 : Handwheel 3 active / Manivelle 3 active
   // // E_Ori[3].HW3 : Handwheel 3 active / Manivelle 3 active
   // // E_Ori[2].TReqMinus : Travel requests minus / Demandes de déplacement moins
   // // E_Ori[3].TReqMinus : Travel requests minus / Demandes de déplacement moins
   // // E_Ori[2].TReqPlus : Travel requests plus / Demandes de déplacement plus
   // // E_Ori[3].TReqPlus : Travel requests plus / Demandes de déplacement plus
   // // E_Ori[2].TCMinus : Traverse command minus / Instruction de déplacement moins
   // // E_Ori[3].TCMinus : Traverse command minus / Instruction de déplacement moins
   // // E_Ori[2].TCPlus : Traverse command plus / Instruction de déplacement plus
   // // E_Ori[3].TCPlus : Traverse command plus / Instruction de déplacement plus
   // // E_Ori[2].INC1 : INC 1 active
   // // E_Ori[3].INC1 : INC 1 active
   // // E_Ori[2].INC10 : INC 10 active
   // // E_Ori[3].INC10 : INC 10 active
   // // E_Ori[2].INC100 : INC 100 active
   // // E_Ori[3].INC100 : INC 100 active
   // // E_Ori[2].INC1000 : INC 1000 active
   // // E_Ori[3].INC1000 : INC 1000 active
   // // E_Ori[2].INC10000 : INC 10000 active
   // // E_Ori[3].INC10000 : INC 10000 active
   // // E_Ori[2].INCVar : INC variable active / Variable INC active
   // // E_Ori[3].INCVar : INC variable active / Variable INC active
   // // E_Ori[2].OEM : OEM signals / Signaux OEM
   // // E_Ori[3].OEM : OEM signals / Signaux OEM
   // // E_Ori[2].InvHWDirOfRot : Handwheel direction of rotation invert actively / Inverser activement sens manivelle
   // // E_Ori[3].InvHWDirOfRot : Handwheel direction of rotation invert actively / Inverser activement sens manivelle
   // // E_Ori[1] : Control signals for orientation axes [1..3] / Signaux de commande pour axes d'orientation [1..3]
   // // E_Ori[2] : Control signals for orientation axes [1..3] / Signaux de commande pour axes d'orientation [1..3]
   // // E_Ori[3] : Control signals for orientation axes [1..3] / Signaux de commande pour axes d'orientation [1..3]
END_TYPE
